// TwinCAT 3 PLC project XyTable
// ProgramVersion: 3.1.4023.0
// libraries:
//   Struckig, 0.12.2.0 (Stefan Besler)
//   Tc2_Standard, * (Beckhoff Automation GmbH)
//   Tc3_Module, 3.4.5.0 (Beckhoff Automation GmbH)
//   ZApplication, 1.5.38.0 (Zeugwerk GmbH)
//   ZAux, 1.5.38.0 (Zeugwerk GmbH)
//   ZCore, 1.5.38.0 (Zeugwerk GmbH)
//   ZEquipment, 1.5.38.0 (Zeugwerk GmbH)
//   ZPlatform, 1.5.38.0 (Zeugwerk GmbH)
// project tree:
//   ZApp/App/ ZApp.TcPOU
//   ZApp/App/_DataTypes/ ZAppStep.TcDUT
//   ZApp/App/_States/ ZAppSequenceBoot.TcPOU, ZAppSequenceBootFault.TcPOU, ZAppSequenceRunning.TcPOU
//   ZApp/App/_SubObjects/ ZAppSequence.TcPOU
//   ZApp/Com/_DataTypes/ ZCom.TcDUT, ZComUnit.TcDUT
//   ZApp/Data/_DataTypes/ ZData.TcDUT, ZDataMachine.TcDUT, ZDataConfig.TcDUT, ZDataCalibration.TcDUT, ZDataRecipe.TcDUT
//   ZApp/Unit/XyTable/ IXyTable.TcIO, XyTableUnit.TcPOU, XyTableUnitProgram.TcPOU
//   ZApp/Unit/XyTable/Segments/ RingBufferSegment.TcPOU (not stored), Segment.TcDUT (not stored), SegmentType.TcDUT (not stored)
//   ZApp/Unit/XyTable/_Com/ XyTableComSubscribeSegments.TcDUT, XyTableCom.TcDUT, XyTableComPublish.TcDUT, XyTableComPublishEquipment.TcDUT, XyTableComRef.TcDUT, XyTableComRequest.TcDUT, XyTableComSubscribe.TcDUT, XyTableComSubscribeEquipment.TcDUT
//   ZApp/Unit/XyTable/_DataTypes/ XyTableState.TcDUT, XyTableStep.TcDUT
//   ZApp/Unit/XyTable/_Data/ XyTableDataCalibration.TcDUT, XyTableDataConfig.TcDUT, XyTableDataMachine.TcDUT, XyTableDataRef.TcDUT
//   ZApp/Unit/XyTable/_Equipment/ XyTableActuator.TcPOU, XyTableActuatorPen.TcPOU, XyTableAxis.TcPOU, XyTableEquipment.TcPOU, XyTableFieldbus.TcPOU, XyTableIo.TcPOU, XyTableLinkedUnit.TcPOU
//   ZApp/Unit/XyTable/_States/ XyTableSequenceAutomatic.TcPOU, XyTableSequenceBoot.TcPOU, XyTableSequenceFaultReaction.TcPOU, XyTableSequenceGoHome.TcPOU, XyTableSequenceStop.TcPOU
//   ZApp/Unit/XyTable/_SubObjects/ XyTableContainer.TcPOU, XyTableSequence.TcPOU
//   ZApp/ ZGlobal.TcGVL, ZModuleProgram.TcPOU, ZModuleTask.TcTTO
// real-time tasks:
//   TASK ZModuleTask: cycle T#10ms, priority 20, ADS port 350

CONFIGURATION XyTable
    RESOURCE PLC ON TwinCAT3
        TASK ZModuleTask(INTERVAL := T#1ms, PRIORITY := 20);
        PROGRAM ZModuleProgram WITH ZModuleTask : ZModuleProgram;
    END_RESOURCE
END_CONFIGURATION

// ---- ZApp/App/_DataTypes/ZAppStep.TcDUT
{attribute 'qualified_only'}
{attribute 'to_string'}
TYPE ZAppStep :
(
  Undefined := 0
  
  ,BootBegin
  ,BootLoadDefaultData
  ,BootEnd
  ,BootFaultBegin
  ,BootFaultEnd 
  ,RunningBegin
  ,RunningEnd   
);
END_TYPE

// ---- ZApp/Com/_DataTypes/ZCom.TcDUT
TYPE ZCom :
STRUCT
  // module context
  App : ZApplication.ApplicationComPublish;
  Alarming : ZApplication.AlarmingCom;
  Messages : ZApplication.MessagingCom;
  
  // unit context
  Unit : ZComUnit;

END_STRUCT
END_TYPE

// ---- ZApp/Com/_DataTypes/ZComUnit.TcDUT
TYPE ZComUnit :
STRUCT
{region "XyTable"}
{IF NOT (defined (XyTable_disabled))}
  XyTable : XyTableCom;
  {attribute 'ZId' := '934662f7-81a9-4247-b804-76d465c7ec61'}
{END_IF}
{endregion}
{attribute '__ZwPlcApplicationComUnitDeclaration__'} // Do not remove this attribute! It is used for code generation.
END_STRUCT
END_TYPE

// ---- ZApp/Data/_DataTypes/ZData.TcDUT
TYPE ZData :
STRUCT
  Config : ZDataConfig;
  Machine : ZDataMachine;
  Calibration : ZDataCalibration;
  Recipe : ZDataRecipe;
END_STRUCT
END_TYPE

// ---- ZApp/Data/_DataTypes/ZDataMachine.TcDUT
TYPE ZDataMachine :
STRUCT
{region "XyTable"}
{IF NOT (defined (XyTable_disabled))}
  XyTable : XyTableDataMachine;
  {attribute 'ZId' := '934662f7-81a9-4247-b804-76d465c7ec61'}
{END_IF}
{endregion}
{attribute '__ZwPlcApplicationDataMachineDeclaration__'} // Do not remove this attribute! It is used for code generation.
END_STRUCT
END_TYPE

// ---- ZApp/Data/_DataTypes/ZDataConfig.TcDUT
TYPE ZDataConfig :
STRUCT
{region "XyTable"}
{IF NOT (defined (XyTable_disabled))}
  XyTable : XyTableDataConfig;
  {attribute 'ZId' := '934662f7-81a9-4247-b804-76d465c7ec61'}
{END_IF}
{endregion}
{attribute '__ZwPlcApplicationDataConfigDeclaration__'} // Do not remove this attribute! It is used for code generation.
END_STRUCT
END_TYPE

// ---- ZApp/Data/_DataTypes/ZDataCalibration.TcDUT
TYPE ZDataCalibration :
STRUCT
{region "XyTable"}
{IF NOT (defined (XyTable_disabled))}
  XyTable : XyTableDataCalibration;
  {attribute 'ZId' := '934662f7-81a9-4247-b804-76d465c7ec61'}
{END_IF}
{endregion}
{attribute '__ZwPlcApplicationDataCalibrationDeclaration__'} // Do not remove this attribute! It is used for code generation.
END_STRUCT
END_TYPE

// ---- ZApp/Data/_DataTypes/ZDataRecipe.TcDUT
TYPE ZDataRecipe :
STRUCT
  RecipeParam1 : LREAL;
  RecipeParam2 : LREAL;
  RecipeParam3 : LREAL;
END_STRUCT
END_TYPE

// ---- ZApp/Unit/XyTable/_Com/XyTableComSubscribeSegments.TcDUT
TYPE XyTableComSubscribeSegments :
STRUCT
  Start : DINT;
  End : DINT;
  Data : ARRAY[0..200] OF Segment;
END_STRUCT
END_TYPE

// ---- ZApp/Unit/XyTable/_Com/XyTableCom.TcDUT
/// This struct contains variables that
/// * are read from outside (e.g. HMI) to retrieve information about the unit's current state and (temporary) parameters (= `publish`) 
/// * are written from outside (e.g. HMI) to control the unit via ADS (= `subscribe`) 
TYPE XyTableCom :
STRUCT
  Publish : XyTableComPublish;
  Subscribe : XyTableComSubscribe;
END_STRUCT
END_TYPE

// ---- ZApp/Unit/XyTable/_Com/XyTableComPublish.TcDUT
/// this is the container of informations that the unit wants to share with the world outside of the PLC
/// This struct should only be read from by external applications.
TYPE XyTableComPublish :
STRUCT
  State : ZApplication.UnitStateMachineState; // state the unit is in
  Request : XyTableComRequest; // booleans that indictate which action is currently possible to perform with this unit
  Equipment : XyTableComPublishEquipment;  // structs for equipment objects which are used by the bridges
END_STRUCT
END_TYPE

// ---- ZApp/Unit/XyTable/_Com/XyTableComPublishEquipment.TcDUT
TYPE XyTableComPublishEquipment :
STRUCT

{region "AxisX : Axis"}
  AxisX : ZApplication.AxisComPublish;
  {attribute 'ZId' := 'fcb4f634-5402-488a-b9f2-f463d25a2352'}
{endregion}

{region "AxisY : Axis"}
  AxisY : ZApplication.AxisComPublish;
  {attribute 'ZId' := '5efb0243-1556-4e56-aeca-16ed0d08aedd'}
{endregion}

{region "Pen : ActuatorDigital"}
  Pen : ZApplication.ActuatorDigitalComPublish;
  PenDown : ZApplication.DigitalComPublish;
  PenUp : ZApplication.DigitalComPublish;
  PenIsDown : ZApplication.DigitalComPublish;
  PenIsUp : ZApplication.DigitalComPublish;
  {attribute 'ZId' := 'a2af64cd-ae98-4060-afd2-2cfacfac101c'}
{endregion}

{attribute '__ZwPlcUnitComDeclaration__'} // Do not remove this attribute! It is used for code generation.

END_STRUCT
END_TYPE

// ---- ZApp/Unit/XyTable/_Com/XyTableComRef.TcDUT
/// container for all communication data types that are used by the unit
TYPE XyTableComRef :
STRUCT
  Publish : REFERENCE TO XyTableComPublish; 
  Subscribe : REFERENCE TO XyTableComSubscribe; 
END_STRUCT
END_TYPE

// ---- ZApp/Unit/XyTable/_Com/XyTableComRequest.TcDUT
TYPE XyTableComRequest :
STRUCT
  Start : BOOL;
  Stop : BOOL;
  GoHome : BOOL;
  Halt : BOOL;
END_STRUCT
END_TYPE

// ---- ZApp/Unit/XyTable/_Com/XyTableComSubscribe.TcDUT
TYPE XyTableComSubscribe :
STRUCT
  Request : XyTableComRequest; // contains booleans that are used to start a specific sequence.
  Equipment : XyTableComSubscribeEquipment;  // structs for equipment objects which are used by the bridges
  Segments : XyTableComSubscribeSegments;
END_STRUCT
END_TYPE

// ---- ZApp/Unit/XyTable/_Com/XyTableComSubscribeEquipment.TcDUT
TYPE XyTableComSubscribeEquipment :
STRUCT

{region "AxisX : Axis"}
  AxisX : ZApplication.AxisComSubscribe;
  {attribute 'ZId' := 'fcb4f634-5402-488a-b9f2-f463d25a2352'}
{endregion}

{region "AxisY : Axis"}
  AxisY : ZApplication.AxisComSubscribe;
  {attribute 'ZId' := '5efb0243-1556-4e56-aeca-16ed0d08aedd'}
{endregion}

{region "Pen : ActuatorDigital"}
  Pen : ZApplication.ActuatorDigitalComSubscribe;
  PenDown : ZApplication.DigitalComSubscribe;
  PenUp : ZApplication.DigitalComSubscribe;
  PenIsDown : ZApplication.DigitalComSubscribe;
  PenIsUp : ZApplication.DigitalComSubscribe;
  {attribute 'ZId' := 'a2af64cd-ae98-4060-afd2-2cfacfac101c'}
{endregion}

{attribute '__ZwPlcUnitComDeclaration__'} // Do not remove this attribute! It is used for code generation.

END_STRUCT
END_TYPE

// ---- ZApp/Unit/XyTable/_DataTypes/XyTableState.TcDUT
/// This enumeration contains all used defined sequences of a unit.
/// Per default a unit makes use of the states that are contained in (UnitStateDefault)[xref:ZApplication.UnitStateDefault]. However,
/// most of the time a unit need to perform some application depend sequences that can be performed by putting the unit into userdefined states.
/// For instance, a robotic unit could use the state (automatic)[xref:ZApplication.UnitStateDefault] to lift an object from point A to point B,
/// a userdefined state could be used to open and close the robotic-units gripper, respectively
{attribute 'qualified_only'}
TYPE XyTableState :
(
	UserdefinedState1 := ZApplication.UnitStateMachineState.Last+1
);
END_TYPE

// ---- ZApp/Unit/XyTable/_DataTypes/XyTableStep.TcDUT
/// This enumeration contains all steps that are used by the various sequences of a unit.
/// Sequences use a subrange (***Begin to ***End) of this enumeration.
{attribute 'qualified_only'}
{attribute 'to_string'}
TYPE XyTableStep :
(
  Undefined := 0
  
  ,BootBegin
  ,BootEnd 

  ,StopBegin
  ,StopEnd

  ,AutomaticBegin
  ,AutomaticWaitSegment
  ,AutomaticMoveToSegmentStart
  ,AutomaticMovePenDown
  ,AutomaticDraw
  ,AutomaticMovePenUp
  ,AutomaticDrawLine
  ,AutomaticDrawCatmulRomDrawSplineBegin
  ,AutomaticDrawCatmulRomDrawSpline
  ,AutomaticEnd
  
  ,GoHomeBegin
  ,GoHomeMoveUp
  ,GoHomeReferenceXY
  ,GoHomeEnd 
  
  ,FaultReactionBegin
  ,FaultReactionEnd
);
END_TYPE

// ---- ZApp/Unit/XyTable/_Data/XyTableDataCalibration.TcDUT
/// calibration that is determined by calibration sequences of the unit (static offsets, shifts)
TYPE XyTableDataCalibration :
STRUCT
END_STRUCT
END_TYPE

// ---- ZApp/Unit/XyTable/_Data/XyTableDataConfig.TcDUT
/// configuration data that is used during boot to configure the Units equipment
TYPE XyTableDataConfig :
STRUCT
  Simulated : BOOL;
END_STRUCT
END_TYPE

// ---- ZApp/Unit/XyTable/_Data/XyTableDataMachine.TcDUT
/// machine data that is used through most sequences of the unit (motor speed, axes positions, ...)
TYPE XyTableDataMachine :
STRUCT
  Slowspeed : LREAL;
  Highspeed : LREAL;
END_STRUCT
END_TYPE

// ---- ZApp/Unit/XyTable/_Data/XyTableDataRef.TcDUT
/// container for all data that are used by the unit
TYPE XyTableDataRef :
STRUCT
  Config : REFERENCE TO XyTableDataConfig; // data required for booting the unit (axes configuration, simulation, parameters that have to be written in PREOP, ...)
  Machine : REFERENCE TO XyTableDataMachine; // speeds, positions, ...
  Calibration : REFERENCE TO XyTableDataCalibration; // offsets, shifts of nominal to actual values
END_STRUCT
END_TYPE

// ---- ZApp/ZGlobal.TcGVL
{attribute 'qualified_only'}
VAR_GLOBAL
  Com : ZCom;
END_VAR
VAR_GLOBAL PERSISTENT
  Data : ZData;
END_VAR

// ---- ZApp/Unit/XyTable/IXyTable.TcIO
INTERFACE IXyTable EXTENDS ZApplication.IUnit

END_INTERFACE

// ---- ZApp/ZModuleProgram.TcPOU
/// Zeugwerk Application
PROGRAM ZModuleProgram
VAR_INPUT
{region "ZModuleProgram : Utility"}
  App : ZApp(displayName:='Zeugwerk-Application Template', com:=ZGlobal.Com.App);
  Datetime : ZAux.DateTimeUM;
  {attribute 'ZId' := ''}
{endregion}
{region "ZModuleProgram : Logging"}
  Alarming : ZApplication.Alarming(App, datetime := Datetime, com := ZGlobal.Com.Alarming);
  LoggerHmi : ZApplication.Messaging(App, datetime := Datetime, com := ZGlobal.Com.Messages);
  LoggerFile : ZAux.LoggerFile7FF(App, datetime := Datetime, filePath:='C:\Zeugwerk\logs\messages.log', target:='');
  Logger : ZAux.Logging;
  {attribute 'ZId' := ''}
{endregion}  
{attribute '__ZwPlcApplicationModuleProgramDeclaration__'} // Do not remove this attribute! It is used for code generation.
{region "XyTable"}
{undefine RunInSeparateProgram}
{IF NOT (defined (XyTable_disabled)) AND NOT (defined (RunInSeparateProgram))}
  XyTable : XyTableUnit(name := 'XyTable', // name of the unit (for logging)
					  parent := App, // caller of the Unit's cyclic method. If the Unit runs in its own context use 0
						configdata := ZGlobal.Data.Config.XyTable,
						machinedata := ZGlobal.Data.Machine.XyTable,
						calibrationdata := ZGlobal.Data.Calibration.XyTable,
						com := ZGlobal.Com.Unit.XyTable);
  {attribute 'section' := '__ZwPlcUnitProgramDeclaration__'}
  {attribute 'ZId' := '934662f7-81a9-4247-b804-76d465c7ec61'}
{END_IF}
{endregion}
{attribute '__ZwPlcUnitProgramDeclaration__'} // Do not remove this attribute! It is used for code generation.
END_VAR

{region "ZModuleProgram : Utility"}
  Datetime.Cyclic();
  App.Cyclic();
  {attribute 'ZId' := ''}
{endregion}
{attribute '__ZwPlcApplicationModuleProgramImplementation__'} // Do not remove this attribute! It is used for code generation.

END_PROGRAM

// ---- ZApp/App/ZApp.TcPOU
FUNCTION_BLOCK ZApp EXTENDS ZApplication.Application
VAR
  _boot : ZAppSequenceBoot;
  _bootFault : ZAppSequenceBootFault;
  _running : ZAppSequenceRunning;
END_VAR

METHOD FB_init : BOOL
VAR_INPUT
  bInitRetains : BOOL; /// if TRUE, the retain variables are initialized (warm start / cold start)
  bInCopyCode : BOOL; /// if TRUE, the instance afterwards gets moved into the copy code (online change)
  displayName : ZCore.ZString;
  com : REFERENCE TO ZApplication.ApplicationComPublish;
END_VAR
SetBootSequence(_boot);
SetBootFaultSequence(_bootFault);
SetRunningSequence(_running);
END_METHOD

END_FUNCTION_BLOCK

// ---- ZApp/App/_States/ZAppSequenceBoot.TcPOU
FUNCTION_BLOCK ZAppSequenceBoot EXTENDS ZAppSequence IMPLEMENTS ZCore.ISequence
VAR
  _step : ZCore.Step(ZAppStep.BootBegin, ZAppStep.BootEnd);
END_VAR

IF OnStart(_step)
THEN
  // init custom sequence variables here ...
END_IF

REPEAT
  LogStep();

  CASE _step.Index OF
    (* -------------------------------------------------------------------------------------------------------------------------------- *)
    ZAppStep.BootBegin:
    (* -------------------------------------------------------------------------------------------------------------------------------- *)
    
      IF _step.OnEntry()
      THEN
        ZModuleProgram.LoggerFile.MinimumLevel := ZCore.LogLevel.Trace;
        ZModuleProgram.Logger.AddLogger(ZModuleProgram.LoggerFile);        
        {attribute '__ZwPlcAppZComModuleContext__'} // Do not remove this attribute! It is used for code generation.      
      END_IF
      
	  IF ZModuleProgram.Datetime.State <> ZCore.ObjectState.Booting
      THEN
        _step.SetNext(ZAppStep.BootLoadDefaultData);        
      END_IF
      
    (* -------------------------------------------------------------------------------------------------------------------------------- *)
    ZAppStep.BootLoadDefaultData:
    (* -------------------------------------------------------------------------------------------------------------------------------- *)

      {warning 'The application is loading the default config data on every restart!'}
      LoadDefaultConfigData();
      
      IF IsCommissioning()
      THEN
        LoadDefaultData();
      END_IF
      
      _step.SetNext(ZAppStep.BootEnd);
      
    (* -------------------------------------------------------------------------------------------------------------------------------- *)
    ZAppStep.BootEnd:
    (* -------------------------------------------------------------------------------------------------------------------------------- *)
      SetBusy(FALSE);
      
  ELSE
    Abort('sequence contains unhandled step');
  END_CASE
UNTIL _step.IsNotRepeatable() OR_ELSE NOT Busy END_REPEAT

METHOD  IsCommissioning : BOOL
IsCommissioning := TRUE;
END_METHOD

METHOD FINAL LoadDefaultConfigData

{region "XyTable"}
  {IF NOT (defined (XyTable_disabled))}
  ZGlobal.Data.Config.XyTable.Simulated := TRUE;
  {region "UserInitCode"}
  // put your individual init code for this unit here
  {endregion}
  {END_IF}
  {attribute 'ZId' := '934662f7-81a9-4247-b804-76d465c7ec61'}
{endregion}

{attribute '__ZwPlcUnitLoadDefaultConfigData__'} // Do not remove this attribute! It is used for code generation.
END_METHOD

METHOD FINAL LoadDefaultData
ZGlobal.Data.Machine.XyTable.Slowspeed := 10;
ZGlobal.Data.Machine.XyTable.Highspeed := 30;

{attribute '__ZwPlcUnitLoadDefaultData__'} // Do not remove this attribute! It is used for code generation.
END_METHOD

END_FUNCTION_BLOCK

// ---- ZApp/App/_SubObjects/ZAppSequence.TcPOU
FUNCTION_BLOCK ABSTRACT ZAppSequence EXTENDS ZApplication.Sequence IMPLEMENTS ZCore.ISequence

METHOD StepDecoded : ZCore.ZString
VAR_INPUT
  stepIndex : INT;
END_VAR
VAR_INST
  _stepIndexDecoded : ZAppStep;
END_VAR
_stepIndexDecoded := stepIndex;
StepDecoded := TO_STRING(_stepIndexDecoded);
END_METHOD

END_FUNCTION_BLOCK

// ---- ZApp/App/_States/ZAppSequenceBootFault.TcPOU
FUNCTION_BLOCK ZAppSequenceBootFault EXTENDS ZAppSequence IMPLEMENTS ZCore.ISequence
VAR
  _step : ZCore.Step(ZAppStep.BootFaultBegin, ZAppStep.BootFaultEnd);
END_VAR

IF OnStart(_step)
THEN
  // init custom sequence variables here ...
END_IF

REPEAT
  LogStep();

  CASE _step.Index OF
    (* -------------------------------------------------------------------------------------------------------------------------------- *)
    ZAppStep.BootFaultBegin:
    (* -------------------------------------------------------------------------------------------------------------------------------- *)
      _step.SetNext(ZAppStep.BootFaultEnd);
      
    (* -------------------------------------------------------------------------------------------------------------------------------- *)
    ZAppStep.BootFaultEnd:
    (* -------------------------------------------------------------------------------------------------------------------------------- *)
      SetBusy(FALSE);
      
  ELSE
    Abort('sequence contains unhandled step');
  END_CASE
UNTIL _step.IsNotRepeatable() OR_ELSE NOT Busy END_REPEAT

END_FUNCTION_BLOCK

// ---- ZApp/App/_States/ZAppSequenceRunning.TcPOU
FUNCTION_BLOCK ZAppSequenceRunning EXTENDS ZAppSequence IMPLEMENTS ZCore.ISequence
VAR
  _step : ZCore.Step(ZAppStep.RunningBegin, ZAppStep.RunningEnd);
END_VAR

IF OnStart(_step)
THEN
  // init custom sequence variables here ...
END_IF

REPEAT
  LogStep();

  CASE _step.Index OF
    (* -------------------------------------------------------------------------------------------------------------------------------- *)
    ZAppStep.RunningBegin:
    (* -------------------------------------------------------------------------------------------------------------------------------- *)
      ; // implement me
      
    (* -------------------------------------------------------------------------------------------------------------------------------- *)
    ZAppStep.RunningEnd:
    (* -------------------------------------------------------------------------------------------------------------------------------- *)
      SetBusy(FALSE);
      
  ELSE
    Abort('sequence contains unhandled step');
  END_CASE
UNTIL _step.IsNotRepeatable() OR_ELSE NOT Busy END_REPEAT

END_FUNCTION_BLOCK

// ---- ZApp/Unit/XyTable/XyTableUnit.TcPOU
/// Declaration of a distinct unit of this application
FUNCTION_BLOCK XyTableUnit EXTENDS ZApplication.Unit IMPLEMENTS IXyTable
VAR
  _equipment : XyTableEquipment(THIS^);
  _data : XyTableDataRef;
  _com : XyTableComRef;

  _boot : XyTableSequenceBoot(THIS^);
  _automatic : XyTableSequenceAutomatic(THIS^);
  _stop : XyTableSequenceStop(THIS^);
  _gohome : XyTableSequenceGoHome(THIS^);
  _faultReaction : XyTableSequenceFaultReaction(THIS^);
  
  _statemachine : ZApplication.UnitStateMachine;

  _observeTimer : ZAux.Timer;
  
  _segments : RingBufferSegment(
                200, 
                ADR(ZGlobal.Com.Unit.XyTable.Subscribe.Segments.Start),
                ADR(ZGlobal.Com.Unit.XyTable.Subscribe.Segments.End),
                ADR(ZGlobal.Com.Unit.XyTable.Subscribe.Segments.Data));      
  
END_VAR

{attribute 'ZId' := '58bf1f70-3606-4d15-9092-18e6bfacf7a1'}

IF _observeTimer.Done THEN
  _observeTimer.WaitAsync(0.1);
  
  // monitor _com for requested actions (e.g. start homing, start automatic mode, ...)
  ObserveRequest(_com.Subscribe.Request.Start, ZApplication.UnitStateMachineState.Automatic);
  ObserveRequest(_com.Subscribe.Request.Stop, ZApplication.UnitStateMachineState.Stop);
  ObserveRequest(_com.Subscribe.Request.GoHome, ZApplication.UnitStateMachineState.GoHome);
  ObserveRequest(_com.Subscribe.Request.Halt, ZApplication.UnitStateMachineState.Halt);
  
  // provide relevant information via ADS
  _com.Publish.Request.Stop := _stateMachine.IsTransitionAllowed(ZApplication.UnitStateMachineState.Stop);
  _com.Publish.Request.Start := _stateMachine.IsTransitionAllowed(ZApplication.UnitStateMachineState.Automatic);
  _com.Publish.Request.GoHome := _stateMachine.IsTransitionAllowed(ZApplication.UnitStateMachineState.GoHome);
  _com.Publish.Request.Halt := _stateMachine.IsTransitionAllowed(ZApplication.UnitStateMachineState.Halt);

  _com.Publish.State := _stateMachine.State();
END_IF

METHOD FB_init : BOOL
VAR_INPUT
  bInitRetains : BOOL; // if TRUE, the retain variables are initialized (warm start / cold start)
  bInCopyCode : BOOL;  // if TRUE, the instance afterwards gets moved into the copy code (online change)
  parent : ZCore.IManagedObject; // caller of the Unit's cyclic method. If the Unit runs in its own context use 0
  name : ZCore.ZString;  // name of this unit as it should show up in the logger
  configdata : REFERENCE TO XyTableDataConfig;  // reference to the configuration data that is used during boot to configure the Units equipment
  machinedata : REFERENCE TO XyTableDataMachine; // reference to the machine data that is used through most sequences of the unit (motor speed, axes positions, ...)
  calibrationdata : REFERENCE TO XyTableDataCalibration;  // reference to calibration that is determined by calibration sequences of the unit (static offsets, shifts)
  com : REFERENCE TO XyTableCom;  // reference to the communication interface that is used to control this Unit via ADS
END_VAR
_name := name;

// initialize local logger decorator
_loggerDecorator.FB_init(bInitRetains, bInCopyCode, name, ZModuleProgram.Logger);
_alarmingDecorator.FB_init(bInitRetains, bInCopyCode, name, ZModuleProgram.Alarming);

// setup data
_data.Config REF= configdata;
_data.Machine REF= machinedata;
_data.Calibration REF= calibrationdata;
_com.Publish REF= com.Publish;
_com.Subscribe REF= com.Subscribe;

// ------- sequence initialization, map sequences of this unit to the statemachine -------
{attribute '__ZwPlcUnitInitSequenceImplementation__'} // Do not remove this attribute! It is used for code generation.
_statemachine.SetSequence(ZApplication.UnitStateMachineState.Boot, _boot);
_statemachine.SetSequence(ZApplication.UnitStateMachineState.FaultReaction, _faultReaction);
_statemachine.SetSequence(ZApplication.UnitStateMachineState.Gohome, _gohome);
_statemachine.SetSequence(ZApplication.UnitStateMachineState.Stop, _stop);
_statemachine.SetSequence(ZApplication.UnitStateMachineState.Automatic, _automatic);

_statemachine.SetName(_name);
_statemachine.SetLogger(_logger);

// set initial state
_statemachine.SetState(ZApplication.UnitStateMachineState.Boot);
SetStateMachine(_statemachine);
END_METHOD

END_FUNCTION_BLOCK

// ---- ZApp/Unit/XyTable/_Equipment/XyTableEquipment.TcPOU
/// This function block is a container for equipment that is used by this unit.
/// Equipment is grouped by its kind (actuator, axes, io, ...).
/// It extends from [ManagedObjectContainer](xref:ZCore.ManagedObjectContainer) such that the parent
/// (= the unit itself) can be passed to equipment instances.
FUNCTION_BLOCK XyTableEquipment EXTENDS XyTableContainer
VAR_INPUT
  Io : XyTableIo(_parent);
  Actuator : XyTableActuator(_parent);
  Axis : XyTableAxis(_parent);
  Fieldbus : XyTableFieldbus(_parent);
  Unit : XyTableLinkedUnit(_parent);
END_VAR

END_FUNCTION_BLOCK

// ---- ZApp/Unit/XyTable/_SubObjects/XyTableContainer.TcPOU
FUNCTION_BLOCK XyTableContainer EXTENDS ZCore.ObjectContainer
VAR_INPUT
END_VAR
VAR_OUTPUT
END_VAR
VAR
  {attribute 'hide'}
  _parent : REFERENCE TO XyTableUnit;
END_VAR

{attribute 'hide' }
METHOD FB_init : BOOL
VAR_INPUT
	bInitRetains : BOOL; // if TRUE, the retain variables are initialized (warm start / cold start)
	bInCopyCode : BOOL;  // if TRUE, the instance afterwards gets moved into the copy code (online change)
  unit : REFERENCE TO XyTableUnit;
END_VAR
_parent REF= unit;
END_METHOD

END_FUNCTION_BLOCK

// ---- ZApp/Unit/XyTable/_Equipment/XyTableIo.TcPOU
/// This function block is a container for all I/Os that are used by this unit.
/// The parent of all objects can be directly transfered in their constructor (this is only relevant for equipment objects
/// that have to be managed (e.g. [DebouncedInput](xref:ZEquipment.DebouncedInput), [Light](xref:ZEquipment.Light), ...).
FUNCTION_BLOCK XyTableIo EXTENDS XyTableContainer
VAR
  {attribute 'hide'}
  _iobridge : ZApplication.IoBridge(_parent);
END_VAR
VAR_INPUT

{attribute '__ZwPlcUnitEquipmentDeclaration__'} // Do not remove this attribute! It is used for code generation.
END_VAR

IF _isInitialized
THEN
  RETURN;
END_IF

  _iobridge.SetLogger(_parent._logger);

{attribute '__ZwPlcUnitEquipmentImplementation__'} // Do not remove this attribute! It is used for code generation.

_isInitialized := TRUE;

END_FUNCTION_BLOCK

// ---- ZApp/Unit/XyTable/_Equipment/XyTableActuator.TcPOU
/// This function block is a container for all actuator objects that are used by this unit.
/// The parent of all objects can be directly transfered in their constructor (this is only relevant for equipment objects
/// that have to be managed (e.g. [DebouncedInput](xref:ZEquipment.DebouncedInput), [Light](xref:ZEquipment.Light), ...).
FUNCTION_BLOCK XyTableActuator EXTENDS XyTableContainer
VAR
  {attribute 'hide'}
  _actuatorbridge : ZApplication.ActuatorBridge(_parent);
  {attribute 'hide'}
  _iobridge : ZApplication.IoBridge(_parent);
END_VAR
VAR_INPUT

{region "Pen : ActuatorDigitalBiLsPlusMinus"}
  Pen : XyTableActuatorPen(_parent);
  {attribute 'ZId' := 'a2af64cd-ae98-4060-afd2-2cfacfac101c'}
{endregion}

{attribute '__ZwPlcUnitEquipmentDeclaration__'} // Do not remove this attribute! It is used for code generation.
END_VAR

IF _isInitialized
THEN
  RETURN;
END_IF

  _actuatorbridge.SetLogger(_parent._logger);

{region "Pen : ActuatorDigitalBiLsPlusMinus"}
  Pen.SetLogger(_parent._logger);
  Pen.SetName(name:='Pen', movePlusName:='Up', moveMinusName:='Down', plusName:='IsUp', minusName:='IsDown');
  Pen.SetSimulation(SEL(_parent._data.Config.Simulated, ActuatorDigitalSimulation.Disabled, ZEquipment.ActuatorDigitalSimulation.Automatic));
  Pen.SetSimulationUncertainty(uncertainty:=0);
  Pen.SetDelay(plusStartDuration:=0, plusEndDuration:=0, minusStartDuration:=0, minusEndDuration:=0, stop:=0);
  Pen.SetSwitchDuration(plusDuration:=0.0, minusDuration:=0.0);
  Pen.SetMovementDuration(plusDuration:=0.75, minusDuration:=0.75);
  Pen.SetTimeout(plusDuration:=5, minusDuration:=5);
  _actuatorbridge.AddActuatorDigital(Pen, publish := _parent._com.Publish.Equipment.Pen, subscribe := _parent._com.Subscribe.Equipment.Pen);
  _iobridge.AddDigitalOutput(Pen.MinusOutput, publish := _parent._com.Publish.Equipment.PenDown, subscribe := _parent._com.Subscribe.Equipment.PenDown);
  _iobridge.AddDigitalOutput(Pen.PlusOutput, publish := _parent._com.Publish.Equipment.PenUp, subscribe := _parent._com.Subscribe.Equipment.PenUp);
  _iobridge.AddDigitalInput(Pen.MinusInput, publish := _parent._com.Publish.Equipment.PenIsDown, subscribe := _parent._com.Subscribe.Equipment.PenIsDown);
  _iobridge.AddDigitalInput(Pen.PlusInput, publish := _parent._com.Publish.Equipment.PenIsUp, subscribe := _parent._com.Subscribe.Equipment.PenIsUp);
  {region "UserInitCode"}
  // put your individual init code for this Actuator here
  {endregion}

  {attribute 'ZId' := 'a2af64cd-ae98-4060-afd2-2cfacfac101c'}
{endregion}

{attribute '__ZwPlcUnitEquipmentImplementation__'} // Do not remove this attribute! It is used for code generation.

_isInitialized := TRUE;

END_FUNCTION_BLOCK

// ---- ZApp/Unit/XyTable/_Equipment/XyTableActuatorPen.TcPOU
FUNCTION_BLOCK XyTableActuatorPen EXTENDS ZEquipment.ActuatorDigitalBiLsPlusMinus

METHOD PUBLIC DownAsync
VAR_INPUT
  startToken : ZCore.IStartToken;
END_VAR
MoveMinusAsync(startToken:=startToken);
END_METHOD

METHOD PUBLIC IsDown : BOOL
VAR_INPUT
END_VAR
IsDown := IsAtMinus();
END_METHOD

METHOD PUBLIC IsUp : BOOL
VAR_INPUT
END_VAR
IsUp := IsAtPlus();
END_METHOD

METHOD PUBLIC UpAsync
VAR_INPUT
  startToken : ZCore.IStartToken;
END_VAR
MovePlusAsync(startToken:=startToken);
END_METHOD

END_FUNCTION_BLOCK

// ---- ZApp/Unit/XyTable/_Equipment/XyTableAxis.TcPOU
/// This function block is a container for all axis objects that are used by this unit.
/// The parent of all objects can be directly transfered in their constructor (this is only relevant for equipment objects
/// that have to be managed (e.g. [DebouncedInput](xref:ZEquipment.DebouncedInput), [Light](xref:ZEquipment.Light), ...).
FUNCTION_BLOCK XyTableAxis EXTENDS XyTableContainer
VAR
  {attribute 'hide'}
  _axisbridge : ZApplication.AxisBridge(_parent);
END_VAR
VAR_INPUT

{region "AxisX : AxisPlcOpenMc"}
  AxisX : ZEquipment.AxisSimulated(_parent);
  {attribute 'ZId' := 'fcb4f634-5402-488a-b9f2-f463d25a2352'}
{endregion}

{region "AxisY : AxisPlcOpenMc"}
  AxisY : ZEquipment.AxisSimulated(_parent);
  {attribute 'ZId' := '5efb0243-1556-4e56-aeca-16ed0d08aedd'}
{endregion}

{attribute '__ZwPlcUnitEquipmentDeclaration__'} // Do not remove this attribute! It is used for code generation.
END_VAR

IF _isInitialized
THEN
  RETURN;
END_IF

  _axisbridge.LoadBalancer.Interval := 0;
  _axisbridge.SetLogger(_parent._logger);

{region "AxisX : AxisPlcOpenMc"}
  AxisX.SetLogger(_parent._logger);
  AxisX.SetName(name:='AxisX');
  AxisX.SetSimulation(_parent._data.Config.Simulated);
  _axisbridge.AddAxisSimulated(axis:=AxisX, publish:=_parent._com.Publish.Equipment.AxisX, subscribe:=_parent._com.Subscribe.Equipment.AxisX);

  {region "UserInitCode"}
  // put your individual init code for this Axis here
  {endregion}

  {attribute 'ZId' := 'fcb4f634-5402-488a-b9f2-f463d25a2352'}
{endregion}

{region "AxisY : AxisPlcOpenMc"}
  AxisY.SetLogger(_parent._logger);
  AxisY.SetName(name:='AxisY');
  AxisY.SetSimulation(_parent._data.Config.Simulated);
  _axisbridge.AddAxisSimulated(axis:=AxisY, publish:=_parent._com.Publish.Equipment.AxisY, subscribe:=_parent._com.Subscribe.Equipment.AxisY);

  {region "UserInitCode"}
  // put your individual init code for this Axis here
  {endregion}

  {attribute 'ZId' := '5efb0243-1556-4e56-aeca-16ed0d08aedd'}
{endregion}

{attribute '__ZwPlcUnitEquipmentImplementation__'} // Do not remove this attribute! It is used for code generation.

_isInitialized := TRUE;

END_FUNCTION_BLOCK

// ---- ZApp/Unit/XyTable/_Equipment/XyTableFieldbus.TcPOU
/// This function block is a container for all axis objects that are used by this unit.
/// The parent of all objects can be directly transfered in their constructor (this is only relevant for equipment objects
/// that have to be managed (e.g. [DebouncedInput](xref:ZEquipment.DebouncedInput), [Light](xref:ZEquipment.Light), ...).
FUNCTION_BLOCK XyTableFieldbus EXTENDS XyTableContainer
VAR
END_VAR
VAR_INPUT

{attribute '__ZwPlcUnitEquipmentDeclaration__'} // Do not remove this attribute! It is used for code generation.
END_VAR

IF _isInitialized
THEN
  RETURN;
END_IF

{attribute '__ZwPlcUnitEquipmentImplementation__'} // Do not remove this attribute! It is used for code generation.

_isInitialized := TRUE;

END_FUNCTION_BLOCK

// ---- ZApp/Unit/XyTable/_Equipment/XyTableLinkedUnit.TcPOU
/// This function block is a container for all linked units that are used by this unit.
/// Linked units can be addressed through their individual interface.
FUNCTION_BLOCK XyTableLinkedUnit EXTENDS XyTableContainer
VAR_INPUT

{attribute '__ZwPlcUnitEquipmentDeclaration__'} // Do not remove this attribute! It is used for code generation.
END_VAR

IF _isInitialized
THEN
  RETURN;
END_IF

{attribute '__ZwPlcUnitEquipmentImplementation__'} // Do not remove this attribute! It is used for code generation.

_isInitialized := TRUE;

END_FUNCTION_BLOCK

// ---- ZApp/Unit/XyTable/_States/XyTableSequenceBoot.TcPOU
FUNCTION_BLOCK XyTableSequenceBoot EXTENDS XyTableSequence IMPLEMENTS ZCore.ISequence
VAR
  _step : ZCore.Step(XyTableStep.BootBegin, XyTableStep.BootEnd);
END_VAR

IF OnStart(_step) THEN
  ; // init custom sequence variables here ...
END_IF

REPEAT
  LogStep();

  CASE _step.Index OF
    (* -------------------------------------------------------------------------------------------------------------------------------- *)
    XyTableStep.BootBegin:
    (* -------------------------------------------------------------------------------------------------------------------------------- *)
      IF _step.OnEntry()
      THEN
        // initialize equipment
        _io();
        _actuator();
        _fieldbus();
        _axis();
        _unit();
      END_IF
      
      _parent._objectManager.Cyclic();      
      Assert(_parent._objectManager);
      IF _parent._objectManager.Booted
      THEN
        _step.SetNext(XyTableStep.BootEnd);
      END_IF

    (* -------------------------------------------------------------------------------------------------------------------------------- *)
    XyTableStep.BootEnd:
    (* -------------------------------------------------------------------------------------------------------------------------------- *)
      SetBusy(FALSE);
      
  ELSE
    Abort('sequence contains unhandled step');
  END_CASE
UNTIL _step.IsNotRepeatable() OR_ELSE NOT Busy END_REPEAT

END_FUNCTION_BLOCK

// ---- ZApp/Unit/XyTable/_SubObjects/XyTableSequence.TcPOU
FUNCTION_BLOCK XyTableSequence EXTENDS ZApplication.Sequence
VAR
  {attribute 'hide'}
  _parent : REFERENCE TO XyTableUnit;
  _io : REFERENCE TO XyTableIo;
  _actuator : REFERENCE TO XyTableActuator;
  _fieldbus : REFERENCE TO XyTableFieldbus;
  _axis : REFERENCE TO XyTableAxis;
  _data : REFERENCE TO XyTableDataRef;
  _unit : REFERENCE TO XyTableLinkedUnit;
  _segments : REFERENCE TO RingBufferSegment;
END_VAR

METHOD FB_init : BOOL
VAR_INPUT
  bInitRetains : BOOL; // if TRUE, the retain variables are initialized (warm start / cold start)
  bInCopyCode : BOOL;  // if TRUE, the instance afterwards gets moved into the copy code (online change)
  unit : REFERENCE TO XyTableUnit;
END_VAR
_parent REF= unit;
_alarming := unit._alarming;
_io REF= unit._equipment.Io;
_actuator REF= unit._equipment.Actuator;
_fieldbus REF= unit._equipment.Fieldbus;
_axis REF= unit._equipment.Axis;
_unit REF= unit._equipment.Unit;
_data REF= unit._data;
_loggerDiagnostics.SetLogger(unit._logger);

_segments REF= unit._segments;
END_METHOD

METHOD StepDecoded : ZCore.ZString
VAR_INPUT
  stepIndex : INT;
END_VAR
VAR_INST
  _stepIndexDecoded : XyTableStep;
END_VAR
_stepIndexDecoded := stepIndex;
stepDecoded := TO_STRING(_stepIndexDecoded);
END_METHOD

END_FUNCTION_BLOCK

// ---- ZApp/Unit/XyTable/_States/XyTableSequenceAutomatic.TcPOU
FUNCTION_BLOCK XyTableSequenceAutomatic EXTENDS XyTableSequence IMPLEMENTS ZCore.ISequence
VAR
  _step : ZCore.Step(XyTableStep.AutomaticBegin, XyTableStep.AutomaticEnd);
  _segment : REFERENCE TO Segment;
  _rt : ZAux.RealTime;
  _otg : Struckig.Otg(0.001, 2);
  
  _splineLogicBuffer : ARRAY [0..8] OF DINT;
  _splinePointBuffer : ARRAY [0..8*2] OF LREAL;
  _splineTangentBuffer : ARRAY [0..8*2] OF LREAL;
  _splineSegmentBuffer : ARRAY [0..8] OF LREAL;
  _spline : ZCore.CatmullRomSpline(8, ADR(_splineLogicBuffer), ADR(_splinePointBuffer), ADR(_splineTangentBuffer), ADR(_splineSegmentBuffer), 2);
  
  _splineIndex : INT;
  i : INT;
END_VAR
VAR_OUTPUT
  ProbeX : LREAL;
  ProbeY : LREAL;
END_VAR

IF NOT Busy THEN
  RETURN;
END_IF

IF OnStart(_step) THEN
  ; // init custom sequence variables here ...
END_IF

IF OnStop() THEN
  RETURN; // external stop was triggered
END_IF

IF OnHalt() THEN
  Halting := TRUE; // Uncomment to acknowledge that the sequence is halting
END_IF

REPEAT
  LogStep();

  CASE _step.Index OF
    (* -------------------------------------------------------------------------------------------------------------------------------- *)
    XyTableStep.AutomaticBegin:
    (* -------------------------------------------------------------------------------------------------------------------------------- *)
      IF _step.OnEntry()
      THEN
        _axis.AxisX.MoveInterpolatedPositionAsync(THIS^);
        _axis.AxisY.MoveInterpolatedPositionAsync(THIS^); 
      END_IF

      Await2(_axis.AxisX, _axis.AxisY, XyTableStep.AutomaticWaitSegment);
    
    (* -------------------------------------------------------------------------------------------------------------------------------- *)
    XyTableStep.AutomaticWaitSegment:
    (* -------------------------------------------------------------------------------------------------------------------------------- *)
      IF _step.OnEntry()
      THEN
        Milestone('Waiting for segment');
              
        _otg.CycleTime := _rt.CycleTimeInSeconds();
        _otg.ControlInterface := Struckig.ControlInterfaceType.Position;
        _otg.Discretization := Struckig.DiscretizationType.Discrete;
        _otg.EnableAutoPropagate := TRUE;  
        _otg.Synchronization := Struckig.SynchronizationType.Phase;        
        _otg.MaxJerk[0] := 100000;
        _otg.MaxJerk[1] := 100000;         
        _otg.MaxAcceleration[0] := 10000;
        _otg.MaxAcceleration[1] := 10000; 
        _otg.MaxVelocity[0] := _data.Machine.Highspeed;
        _otg.MaxVelocity[1] := _data.Machine.Highspeed;
      END_IF

      IF Halting
      THEN
        _step.SetNext(XyTableStep.AutomaticEnd);
      ELSIF NOT _segments.Empty
      THEN
        _segment REF= _segments.ItemAt(0);
        _step.SetNext(XyTableStep.AutomaticMoveToSegmentStart);
			END_IF


    (* -------------------------------------------------------------------------------------------------------------------------------- *)
    XyTableStep.AutomaticMoveToSegmentStart:
    (* -------------------------------------------------------------------------------------------------------------------------------- *)
      IF _step.OnEntry()
      THEN
        _otg.TargetPosition[0] := _segment.Points[0].X;
        _otg.TargetPosition[1] := _segment.Points[0].Y;      
        _otg.TargetVelocity[0] := 0; 
        _otg.TargetVelocity[1] := 0;      
      ELSIF _otg.State = Struckig.TrajectoryState.Idle
      THEN
        _step.SetNext(XyTableStep.AutomaticMovePenDown);
      END_IF

    
    (* -------------------------------------------------------------------------------------------------------------------------------- *)
    XyTableStep.AutomaticMovePenDown:
    (* -------------------------------------------------------------------------------------------------------------------------------- *)
      IF _step.OnEntry()
      THEN
        _actuator.Pen.DownAsync(THIS^);
      END_IF

      Await(_actuator.Pen, XyTableStep.AutomaticDraw);

    (* -------------------------------------------------------------------------------------------------------------------------------- *)
    XyTableStep.AutomaticDraw:
    (* -------------------------------------------------------------------------------------------------------------------------------- *)
      
      CASE _segment.Verb
      OF
        SegmentType.LinePoints: _step.SetNext(XyTableStep.AutomaticDrawLine);
        SegmentType.CatmulRomPoints: _step.SetNext(XyTableStep.AutomaticDrawCatmulRomDrawSplineBegin);
      ELSE
        Abort('Unsupported Verb');     
      END_CASE
      
    (* -------------------------------------------------------------------------------------------------------------------------------- *)
    XyTableStep.AutomaticMovePenUp:
    (* -------------------------------------------------------------------------------------------------------------------------------- *)
      IF _step.OnEntry()
      THEN
      
        _segments.PopFirstItem();
        
        IF _segments.Empty
          OR_ELSE NOT ZCore.IsEqualLreal(_otg.CurrentPosition[0], _segments.ItemAt(0).Points[0].X, 0.1) 
          OR_ELSE NOT ZCore.IsEqualLreal(_otg.CurrentPosition[1], _segments.ItemAt(0).Points[0].Y, 0.1)
        THEN
          _actuator.Pen.UpAsync(THIS^);
        END_IF 
      END_IF

      Await(_actuator.Pen, XyTableStep.AutomaticWaitSegment);
      
    (* -------------------------------------------------------------------------------------------------------------------------------- *)
    XyTableStep.AutomaticDrawLine:
    (* -------------------------------------------------------------------------------------------------------------------------------- *)
      IF _step.OnEntry()
      THEN
        _otg.CurrentAcceleration[0] := 0;
        _otg.CurrentAcceleration[1] := 0;
        _otg.CurrentVelocity[0] := 0;
        _otg.CurrentVelocity[1] := 0;        
        _otg.CurrentPosition[0] := _segment.Points[0].X;
        _otg.CurrentPosition[1] := _segment.Points[0].Y;
        _otg.TargetPosition[0] := _segment.Points[1].X;
        _otg.TargetPosition[1] := _segment.Points[1].Y;        
        _otg.TargetAcceleration[0] := 0;
        _otg.TargetAcceleration[1] := 0;
        _otg.TargetVelocity[0] := 0;
        _otg.TargetVelocity[1] := 0;
      ELSIF _otg.State = Struckig.TrajectoryState.Idle
      THEN
        _step.SetNext(XyTableStep.AutomaticMovePenUp);        
			END_IF

    (* -------------------------------------------------------------------------------------------------------------------------------- *)
    XyTableStep.AutomaticDrawCatmulRomDrawSplineBegin:
    (* -------------------------------------------------------------------------------------------------------------------------------- *)
    
      _otg.CycleTime := _rt.CycleTimeInSeconds();
      _otg.ControlInterface := Struckig.ControlInterfaceType.Position;
      _otg.Discretization := Struckig.DiscretizationType.Discrete;
      _otg.EnableAutoPropagate := TRUE;
      _otg.Synchronization := Struckig.SynchronizationType.Phase;    
      _otg.CurrentAcceleration[0] := 0;
      _otg.CurrentAcceleration[1] := 0;        
      _otg.CurrentVelocity[0] := 0;
      _otg.CurrentVelocity[1] := 0;        
      _otg.CurrentPosition[0] := _segment.Points[0].X;
      _otg.CurrentPosition[1] := _segment.Points[0].Y;
      _otg.TargetAcceleration[0] := 0;
      _otg.TargetAcceleration[1] := 0;  
      _spline.Clear();
      
      // todo: make this more dynamic ...
      FOR i:=0 TO 4
      DO 
        _spline.Append(((i) / INT_TO_LREAL(4)), ADR(_segment.Points[i]));
      END_FOR

      _spline.Interpolate(0,0,0,0);
      _splineIndex := 0;
      _step.SetNext(XyTableStep.AutomaticDrawCatmulRomDrawSpline);
      

    (* -------------------------------------------------------------------------------------------------------------------------------- *)
    XyTableStep.AutomaticDrawCatmulRomDrawSpline:
    (* -------------------------------------------------------------------------------------------------------------------------------- *)
      IF _step.OnEntry()
      THEN
        _otg.TargetPosition[0] := _splinePointBuffer[_splineIndex*2];
        _otg.TargetPosition[1] := _splinePointBuffer[_splineIndex*2+1];      
        _otg.TargetVelocity[0] := _splineTangentBuffer[_splineIndex*2+1]; 
        _otg.TargetVelocity[1] := _splineTangentBuffer[_splineIndex*2+1]; 
      ELSIF _otg.State = Struckig.TrajectoryState.Idle
      THEN
        IF _splineIndex < 4
        THEN
          _splineIndex := _splineIndex + 1;
          _step.RepeatStep();
        ELSE
          _step.SetNext(XyTableStep.AutomaticMovePenUp);                  
				END_IF
			END_IF      
    
    (* -------------------------------------------------------------------------------------------------------------------------------- *)
    XyTableStep.AutomaticEnd:
    (* -------------------------------------------------------------------------------------------------------------------------------- *)
      SetBusy(FALSE);
  
  ELSE
    Abort('sequence contains unhandled step');
  END_CASE
UNTIL _step.IsNotRepeatable() OR_ELSE NOT Busy END_REPEAT

IF _step.Index >= XyTableStep.AutomaticWaitSegment
THEN
  _otg();
  
  IF _otg.State = Struckig.TrajectoryState.Error
  THEN
    Abort(_otg.ErrorMessage());
  ELSE
    _axis.AxisX.SetInterpolatedPosition(THIS^, _otg.CurrentPosition[0]);
    _axis.AxisY.SetInterpolatedPosition(THIS^, _otg.CurrentPosition[1]);
    _axis.AxisX.SetInterpolatedVelocity(THIS^, _otg.CurrentVelocity[0]);
    _axis.AxisY.SetInterpolatedVelocity(THIS^, _otg.CurrentVelocity[1]);    
	END_IF

END_IF

END_FUNCTION_BLOCK

// ---- ZApp/Unit/XyTable/_States/XyTableSequenceStop.TcPOU
FUNCTION_BLOCK XyTableSequenceStop EXTENDS XyTableSequence IMPLEMENTS ZCore.ISequence
VAR
  _step : ZCore.Step(XyTableStep.StopBegin, XyTableStep.StopEnd);
  _timerSim : ZAux.Timer;
END_VAR

IF OnStart(_step) THEN
  ; // init custom sequence variables here ...
END_IF

REPEAT
  LogStep();

  CASE _step.Index OF
    (* -------------------------------------------------------------------------------------------------------------------------------- *)
    XyTableStep.StopBegin:
    (* -------------------------------------------------------------------------------------------------------------------------------- *)
      IF _step.OnEntry()
      THEN
        _actuator.Pen.UpAsync(THIS^);
        _axis.AxisX.StopAsync(THIS^);
        _axis.AxisY.StopAsync(THIS^);
			END_IF
      
      Await3(_actuator.Pen, _axis.AxisX, _axis.AxisY, nextStep:=XyTableStep.StopEnd);

    (* -------------------------------------------------------------------------------------------------------------------------------- *)
    XyTableStep.StopEnd:
    (* -------------------------------------------------------------------------------------------------------------------------------- *)    
      SetBusy(FALSE);
  
  ELSE
    Abort('sequence contains unhandled step');
  END_CASE
UNTIL _step.IsNotRepeatable() OR_ELSE NOT Busy END_REPEAT

END_FUNCTION_BLOCK

// ---- ZApp/Unit/XyTable/_States/XyTableSequenceGoHome.TcPOU
FUNCTION_BLOCK XyTableSequenceGoHome EXTENDS XyTableSequence IMPLEMENTS ZCore.ISequence
VAR
  _step : ZCore.Step(XyTableStep.GohomeBegin, XyTableStep.GohomeEnd);
  _timer : ZAux.Timer;
END_VAR

IF NOT Busy THEN
  RETURN;
END_IF

IF OnStart(_step) THEN
  ; // init custom sequence variables here ...
END_IF

IF OnStop() THEN
  RETURN; // external stop was triggered
END_IF

IF OnHalt() THEN
  ; // Halting := TRUE; // Uncomment to acknowledge that the sequence is halting
END_IF

REPEAT
  LogStep();

  CASE _step.Index OF
    (* -------------------------------------------------------------------------------------------------------------------------------- *)
    XyTableStep.GoHomeBegin:
    (* -------------------------------------------------------------------------------------------------------------------------------- *)
      IF _step.OnEntry()
      THEN
        ;
			END_IF

      _step.SetNext(index:=XyTableStep.GoHomeMoveUp);

    (* -------------------------------------------------------------------------------------------------------------------------------- *)
    XyTableStep.GoHomeMoveUp:
    (* -------------------------------------------------------------------------------------------------------------------------------- *)
      IF _step.OnEntry()
      THEN
        _actuator.Pen.UpAsync(THIS^);
			END_IF
      
      Await(_actuator.Pen, nextStep:=XyTableStep.GoHomeReferenceXY);

    (* -------------------------------------------------------------------------------------------------------------------------------- *)
    XyTableStep.GoHomeReferenceXY:
    (* -------------------------------------------------------------------------------------------------------------------------------- *)
      IF _step.OnEntry()
      THEN
        _axis.AxisX.HomingAsync(THIS^);
        _axis.AxisY.HomingAsync(THIS^);
			END_IF
      
      Await3(_actuator.Pen, _axis.AxisX, _axis.AxisY, nextStep:=XyTableStep.GoHomeEnd);

    (* -------------------------------------------------------------------------------------------------------------------------------- *)
    XyTableStep.GoHomeEnd:
    (* -------------------------------------------------------------------------------------------------------------------------------- *)
      SetBusy(FALSE);
  
  ELSE
    Abort('sequence contains unhandled step');
  END_CASE
UNTIL _step.IsNotRepeatable() OR_ELSE NOT Busy END_REPEAT

END_FUNCTION_BLOCK

// ---- ZApp/Unit/XyTable/_States/XyTableSequenceFaultReaction.TcPOU
FUNCTION_BLOCK XyTableSequenceFaultReaction EXTENDS XyTableSequence IMPLEMENTS ZCore.ISequence
VAR
  _step : ZCore.Step(XyTableStep.FaultReactionBegin, XyTableStep.FaultReactionEnd);
  _timer : ZAux.Timer;
END_VAR

IF OnStart(_step) THEN
  ; // init custom sequence variables here ...
END_IF

REPEAT
  LogStep();

  CASE _step.Index OF
    (* -------------------------------------------------------------------------------------------------------------------------------- *)
    XyTableStep.FaultReactionBegin:
    (* -------------------------------------------------------------------------------------------------------------------------------- *)
      IF _step.OnEntry()
      THEN
        _actuator.Pen.UpAsync(THIS^);
        _axis.AxisX.StopAsync(THIS^);
        _axis.AxisY.StopAsync(THIS^);
        _timer.WaitAsync(2);
			END_IF
      
      Await3(_actuator.Pen, _axis.AxisX, _axis.AxisY, nextStep:=XyTableStep.FaultReactionEnd);
      IF _timer.Done
      THEN
        _step.SetNext(XyTableStep.FaultReactionEnd);
			END_IF

    (* -------------------------------------------------------------------------------------------------------------------------------- *)
    XyTableStep.FaultReactionEnd:
    (* -------------------------------------------------------------------------------------------------------------------------------- *)    
      SetBusy(FALSE);
  
  ELSE
    Abort('sequence contains unhandled step');
  END_CASE
UNTIL _step.IsNotRepeatable() OR_ELSE NOT Busy END_REPEAT

END_FUNCTION_BLOCK

// ---- ZApp/Unit/XyTable/XyTableUnitProgram.TcPOU
/// each unit can run in its own PROGRAM and Task, respectively. However, this is optional and one may also
/// instantiate the unit in the ModuleProgram.
/// In order to keep initialization to a minimum, all ModuleContext objects that are required by the Unit are
/// given as FB_init parameter. These objects are
/// * data structs
/// * communication structs
/// * busmaster(s)
/// A unit should always be a root object (no parent) if it is running in its own context. If it runs in the same
/// task as the Module the parent may be set to the Module's Application.
PROGRAM XyTableUnitProgram
VAR
{region "XyTable"}
{undefine RunInSeparateProgram}
{IF NOT (defined (XyTable_disabled)) AND (defined (RunInSeparateProgram))}
  XyTable : XyTableUnit(name := 'XyTable', // name of the unit (for logging)
					  parent := 0, // caller of the Unit's cyclic method. If the Unit runs in its own context use 0
						configdata := ZGlobal.Data.Config.XyTable,
						machinedata := ZGlobal.Data.Machine.XyTable,
						calibrationdata := ZGlobal.Data.Calibration.XyTable,
						com := ZGlobal.Com.Unit.XyTable);
  {attribute 'section' := '__ZwPlcUnitProgramDeclaration__'}
  {attribute 'ZId' := '934662f7-81a9-4247-b804-76d465c7ec61'}
{END_IF}
{endregion}
{attribute '__ZwPlcUnitProgramDeclaration__'} // Do not remove this attribute! It is used for code generation.
END_VAR

// run the unit - the cylics of all children will be called as well

{region "XyTable"}
{undefine RunInSeparateProgram}
{IF NOT (defined (XyTable_disabled)) AND (defined (RunInSeparateProgram))}
  XyTable.Cyclic();
  {attribute 'section' := '__ZwPlcUnitProgramImplementation__'}
  {attribute 'ZId' := '934662f7-81a9-4247-b804-76d465c7ec61'}
{END_IF}
{endregion}
{attribute '__ZwPlcUnitProgramImplementation__'} // Do not remove this attribute! It is used for code generation.

END_PROGRAM
